Yaskawa INFORM job: INIT_ROS.JBI

/JOB
//NAME INIT_ROS
//POS
///NPOS 0,0,0,0,0,0
//INST
///DATE 2012/01/01 06:53
///ATTR SC,RW
///GROUP1 RB1
///GROUP2 ST1
NOP
DOUT OT#(889) OFF
DOUT OT#(890) OFF
TIMER T=0.01
DOUT OT#(889) ON
WAIT OT#(890)=ON
DOUT OT#(889) OFF
DOUT OT#(890) OFF
END
